Universal Robots PolyScope program: RC_E7_PICK_720.urp

Program RC_E7_PICK_720 (createdIn=3.0.0 lastSavedIn=3.0.0 directory=/programs installation=default)
Robot Program (runOnlyOnce=true motionType=MoveJ speed=1.047198 acceleration=1.396263 useActiveTCP=false)
  'Program generated by RoboDK v4.1.0 for UR3e_HORNO on 27/07/2022 12:03:07'
  'Using nominal kinematics.'
  'Using Ref. Frame RC Traslado B: p[0.370000, -0.335000, 0.000000, 0.000000, 0.000000, 0.000000]'
  'Using TCP 0208-0001-0001-307-000-3 Horno: p[0.000000, 0.000000, 0.038000, 0.000000, 0.000000, 0.000000]'
  Script: set_tcp(p[0.000000, 0.000000, 0.038000, 0.000000, 0.000000, 0.000000])
  Script: movej([-0.417657, -1.931730, -0.885580, -1.893508, 1.584410, 1.186824],0.60000,0.12500,0,0.0000)
  MoveL speed 100 mm/s, acceleration 120 mm/s^2 (useActiveTCP=true)
    Waypoint Waypoint_1: TCP in base x=651.979 y=-751.335 z=126.748 mm, rx=0.0271 ry=3.1343 rz=0.0181 rad; joints [-40.99, -142.15, -49.85, -78.12, 90.77, 50] deg; flange x=651.705 y=-751.773 z=164.744 mm, rx=0.0271 ry=3.1343 rz=0.0181 rad
  'Attach to 0208-0001-0001-307-000-4 Horno'
  MoveL speed 500 mm/s, acceleration 900 mm/s^2 (useActiveTCP=true)
    Waypoint Waypoint_2: TCP in base x=659.095 y=-604.727 z=317.735 mm, rx=0.0528 ry=3.1343 rz=0.0187 rad; joints [-23.93, -110.68, -50.74, -108.49, 90.78, 68] deg; flange x=658.83 y=-605.176 z=355.732 mm, rx=0.0528 ry=3.1343 rz=0.0187 rad
